// TIA Portal V20 export
TYPE "typeSequenceControlNodeJobInterface_transferPnPRight"
// stored: Namespace Unit1.Em5
   STRUCT
      hipotThicknessPICKJob2 : "LER_typeJobInterface";
      visionPLACEJob3 : "LER_typeJobInterface";
      visionPICKJob4 : "LER_typeJobInterface";
      laserMarkPLACEJob5 : "LER_typeJobInterface";
      laserMarkPICKJob6 : "LER_typeJobInterface";
      weightCheckPLACEJob9 : "LER_typeJobInterface";
   END_STRUCT;
END_TYPE
